FUNCTION_BLOCK FB_RaDecTelescopeControl EXTENDS FB_BaseTelescopeControl IMPLEMENTS I_RaDecTelescope;
VAR_INPUT
END_VAR
VAR_OUTPUT
END_VAR
VAR
	eq2hor				: FB_EQ2HOR;
	hor2eq				: FB_HOR2EQ;

	fHourAngleOffset	: LREAL := 0.0;		// absolute offset for hour angle
	fDeclinationOffset	: LREAL := 0.0;		// absolute offset for declination
	
	fHourAngleVelocity	: LREAL;	// rotational velocity of the HA
	fDeclinationVelocity: LREAL;	// rotational velocity of the declination
	
	fElevationPointing  	: LREAL;	// true position of the elevation with applied pointing model
	fAzimuthPointing    	: LREAL;	// true position of the azimuth with applied pointing model
	fRightAscensionPointing	: LREAL;	// RA from pointing Az/El
	fDeclinationPointing	: LREAL;	// Dec from pointing Az/El
	
	fDerotationSign	: LREAL := 1.0;	// sign of derotation
END_VAR
VAR PERSISTENT
	EOFF				: LREAL;	// elevation encoder zero offset
	AN_E				: LREAL;	// azimuth axis offset/misalignment north-south
	AE_E				: LREAL;	// azimuth axis offset/misalignment east-west
	TF					: LREAL;	// gravitational flexure correction at the horizon
	AOFF				: LREAL;	// azimuth encoder zero offset
	BNP					: LREAL;	// collimation error of the electromagnetic axis
	AN_A				: LREAL;	// azimuth axis offset/misalignment north-south
	AE_A				: LREAL;	// azimuth axis offset/misalignment east-west,
	NPAE				: LREAL;	// Non-perpendicularity between the mount azimuth and elevation axes
END_VAR

SUPER^();

// Alt/Az to RA/Dec
hor2eq(alt := fElevation, 
		az := fAzimuth,
		jd := fJD,
		lat := telescopeConfig.latitude,
		lon := telescopeConfig.longitude,
		altitude := telescopeConfig.altitude,
		ra => fRightAscensionCalc,
		dec => fDeclinationCalc);
		
// to HA
fHourAngleCalc := 0.0;

// apply pointing model
//fRightAscensionCalc := fRightAscensionCalc + PointingModelRightAscension
//fDeclinationCalc := fDeclinationCalc + PointingModelDeclination 

// calculate velocities
//fHourAngleVelocity := F_Elevationvelocity(fAzimuthCalc, telescopeConfig.latitude);
//fDeclinationVelocity := F_Azimuthvelocity(fElevationCalc, fAzimuthCalc, telescopeConfig.latitude);

// apply reverse pointing model
//fElevationPointing := fElevationCurrent - PointingModelElevation(fAzimuthCurrent, fElevationCurrent, EOFF, AN_E, AE_E, TF);
//fAzimuthPointing := fAzimuthCurrent - PointingModelAzimuth(fAzimuthCurrent, fElevationCurrent, AOFF, BNP, AN_A, AE_A, NPAE);

// add offsets
//fElevationCurrent := fElevationPointing - fElevationOffset;
//fAzimuthCurrent := fAzimuthPointing - fAzimuthOffset;

// calculate horizontal coordinates
eq2hor(
	ra := fRightAscensionCurrent,
	dec := fDeclinationCurrent,
	lon := telescopeConfig.longitude,
	lat := telescopeConfig.latitude,
	JD := fJD,
	alt => fElevationCalc,
	az => fAzimuthCalc,
	ha => fHourAngleCalc);

METHOD _PublishTelemetry : BOOL
VAR_INPUT
END_VAR
fbComm.Publish('telescope', 'dome', 'POSITION.INSTRUMENTAL.RA.OFFSET', LREAL_TO_STRING(fHourAngleOffset));
fbComm.Publish('telescope', 'dome', 'POSITION.INSTRUMENTAL.DEC.OFFSET', LREAL_TO_STRING(fDeclinationOffset));
END_METHOD

PROPERTY DeclinationOffset : LREAL
GET
DeclinationOffset := THIS^.fDeclinationOffset;
END_GET
SET
THIS^.fDeclinationOffset := DeclinationOffset;
END_SET
END_PROPERTY

PROPERTY HourAngleOffset : LREAL
GET
HourAngleOffset := THIS^.fHourAngleOffset;
END_GET
SET
THIS^.fHourAngleOffset := HourAngleOffset;
END_SET
END_PROPERTY

END_FUNCTION_BLOCK

(* stored: Version 1.1.0.1, ProductVersion 3.1.4024.15
   POU FB_RaDecTelescopeControl: Id {970d8181-0be4-4e4a-9ab2-2a422d7ff3f2}, SpecialFunc None
   Method _PublishTelemetry: Id {560c4df5-8843-4b45-8467-c2296981790f}
   Property DeclinationOffset: Id {215080a3-42ae-4b14-aacb-d9676be48ca3}
   Get Get: Id {87710857-794a-401d-93b3-bd7eef10dbb4}
   Set Set: Id {e3560324-cc67-4753-8d0b-75a12776739c}
   Property HourAngleOffset: Id {efaf06a9-01bd-4628-be65-b2ee5283ea3f}
   Get Get: Id {cd419ed4-496f-4a4d-8c59-531a86e02332}
   Set Set: Id {e0d989a4-a2a8-47cf-a275-be69780dab82} *)
